FUNCTION ISC_LOWER : BOOL
VAR_INPUT
	IN : BYTE;
END_VAR


(*
version 1.1	19. oct. 2008
programmer 	hugo
tested by	oscat

isc_lower checks if a character is lowercase.

*)

IF setup.EXTENDED_ASCII THEN
	ISC_LOWER := ((in > 96) AND (in < 123)) OR ((in > 222) AND (in <> 247));
ELSE
	ISC_LOWER := ((in > 96) AND (in < 123));
END_IF;

(* revision history
hm	6. mar. 2008	rev 1.0
	original version

hm	19. oct. 2008	rev 1.1
	changes setup constants
*)

END_FUNCTION

(* stored: Version 1.1.0.1, ProductVersion 3.1.4024.9
   POU ISC_LOWER: Id {916118bb-a74d-427b-84eb-3953936d929a}, SpecialFunc None *)
